# EPICS substitutions: evrMrmApp/Db/evr-pcie-300dc.substitutions
# Record set for a PCIe-EVR-300DC
#
# Macros:
#  EVR = Card name (same as mrmEvrSetupPCI())
#  SYS = System name (ie SR-TM)
#  D = Device name (ie EVR:Diag2)
#  FEVT = Event link frequency (default 124.916 MHz)
#
# Record names have the general forms:
#  $(SYS){$(D)}Signal-SD
#  $(SYS){$(D)-SubDev}Signal-SD

file "evrbase.db"
{
{P="$(SYS){$(D)}", PCNT="$(SYS){$(D)}Cnt:", PLINK="$(SYS){$(D)}Link:", PRATE="$(SYS){$(D)}Rate:", PTIME="$(SYS){$(D)}Time:", OBJ="$(EVR)", OBJBUFRX="$(EVR):BUFRX", EVNT1HZ="\$(EVNT1HZ=125)", FEVT="\$(FEVT=124.916)"}
}

file "databuftx.db"
{pattern
{P, OBJ, PROTO}
{"$(SYS){$(D)}dbus:send:", "$(EVR):BUFTX", 1}
}

file "evrSoftEvt.template"
{
{P="$(SYS){$(D)}", OBJ="$(EVR)"}
}

file "databuftxCtrl.db"
{pattern
{P, OBJ}
{"$(SYS){$(D)}Link:", "$(EVR):BUFTX"}
}

file "mrmevrbufrx.db"
{pattern
{P, OBJ, PROTO}
{"$(SYS){$(D)}dbus:recv:", $(EVR):BUFRX, 0xff00}
}

file mrmSoftSeq.template {
pattern { P, PINITSEQ, PTRIGSRC, EVG, seqNum, NELM }
{ "$(SYS){$(D)-SoftSeq:0}", "$(SYS){$(D)-SoftSeq:0}InitSeq:", "$(SYS){$(D)-SoftSeq:0}TrigSrc:", "$(EVR)", 0, 2047 }
{ "$(SYS){$(D)-SoftSeq:1}", "$(SYS){$(D)-SoftSeq:1}InitSeq:", "$(SYS){$(D)-SoftSeq:1}TrigSrc:", "$(EVR)", 1, 2047 }
{ "$(SYS){$(D)-SoftSeq:2}", "$(SYS){$(D)-SoftSeq:2}InitSeq:", "$(SYS){$(D)-SoftSeq:2}TrigSrc:", "$(EVR)", 2, 2047 }
}

file evrSoftSeq.template {
pattern { P, PTRIGSRC, PEVTCLKFREQ, SYSDEVTCLK, EVG, seqNum, NELM }
{ "$(SYS){$(D)-SoftSeq:0}", "$(SYS){$(D)-SoftSeq:0}TrigSrc:", "$(SYS){$(D)-SoftSeq:0}EvtClkFreq:", "$(SYS){$(D)-EvtClk}", "$(EVR)", 0, 2047 }
{ "$(SYS){$(D)-SoftSeq:1}", "$(SYS){$(D)-SoftSeq:1}TrigSrc:", "$(SYS){$(D)-SoftSeq:1}EvtClkFreq:", "$(SYS){$(D)-EvtClk}", "$(EVR)", 1, 2047 }
{ "$(SYS){$(D)-SoftSeq:2}", "$(SYS){$(D)-SoftSeq:2}TrigSrc:", "$(SYS){$(D)-SoftSeq:2}EvtClkFreq:", "$(SYS){$(D)-EvtClk}", "$(EVR)", 2, 2047 }
}

file "sfp.db"
{
{P="$(SYS){$(D)-SFP}", PPWR="$(SYS){$(D)-SFP}Pwr:", PSPEED="$(SYS){$(D)-SFP}Speed:", PDATE="$(SYS){$(D)-SFP}Date:", OBJ="$(EVR):SFP"}
}

file "mrmevrdc.template"
{
{P="$(SYS){$(D)-DC}", OBJ="$(EVR)"}
}

file "evrmap.db"
{pattern
{NAME, OBJ, func, EVT}
{"$(SYS){$(D)}Evt:Blink0-SP", "$(EVR)", Blink, 15}
{"$(SYS){$(D)}Evt:Blink1-SP", "$(EVR)", Blink, 0}
{"$(SYS){$(D)}Evt:ResetPS-SP","$(EVR)", "Reset PS", 123}
}

file "evrevent.db"
{pattern
{EN, OBJ, CODE, EVNT}
{"$(SYS){$(D)}1hz",  "$(EVR)", 0x7d, 125}
{"$(SYS){$(D)}EvtA", "$(EVR)", 10, 10}
{"$(SYS){$(D)}EvtB", "$(EVR)", 11, 11}
{"$(SYS){$(D)}EvtC", "$(EVR)", 12, 12}
{"$(SYS){$(D)}EvtD", "$(EVR)", 13, 13}
{"$(SYS){$(D)}EvtE", "$(EVR)", 14, 14}
{"$(SYS){$(D)}EvtF", "$(EVR)", 15, 15}
{"$(SYS){$(D)}EvtG", "$(EVR)", 16, 16}
{"$(SYS){$(D)}EvtH", "$(EVR)", 17, 17}
}

file "evrscale.db"
{pattern
{IDX, P, SN, OBJ, MAX}
{0, "$(SYS){$(D)}Link:", "$(SYS){$(D)-PS:$(IDX)}", "$(EVR):PS$(IDX)", "0xffffffff"}
{1, "$(SYS){$(D)}Link:", "$(SYS){$(D)-PS:$(IDX)}", "$(EVR):PS$(IDX)", "0xffffffff"}
{2, "$(SYS){$(D)}Link:", "$(SYS){$(D)-PS:$(IDX)}", "$(EVR):PS$(IDX)", "0xffffffff"}
{3, "$(SYS){$(D)}Link:", "$(SYS){$(D)-PS:$(IDX)}", "$(EVR):PS$(IDX)", "0xffffffff"}
{4, "$(SYS){$(D)}Link:", "$(SYS){$(D)-PS:$(IDX)}", "$(EVR):PS$(IDX)", "0xffffffff"}
{5, "$(SYS){$(D)}Link:", "$(SYS){$(D)-PS:$(IDX)}", "$(EVR):PS$(IDX)", "0xffffffff"}
{6, "$(SYS){$(D)}Link:", "$(SYS){$(D)-PS:$(IDX)}", "$(EVR):PS$(IDX)", "0xffffffff"}
{7, "$(SYS){$(D)}Link:", "$(SYS){$(D)-PS:$(IDX)}", "$(EVR):PS$(IDX)", "0xffffffff"}
}

file "mrmevrout.db"
{pattern
{ON, ONSRC, OBJ, DESC}
{"$(SYS){$(D)-Out:Int}", "$(SYS){$(D)-Out:Int}Src:", "$(EVR):Int", "Internal"}
# default to tri-state for IFB
pattern
{ON, ONSRC, OBJ, DESC, DEFAULT}
{"$(SYS){$(D)-Out:FPUV00}", "$(SYS){$(D)-Out:FPUV00}Src:", "$(EVR):FrontUnivOut0", "UNIV0", 61}
{"$(SYS){$(D)-Out:FPUV01}", "$(SYS){$(D)-Out:FPUV01}Src:", "$(EVR):FrontUnivOut1", "UNIV1", 61}
{"$(SYS){$(D)-Out:FPUV02}", "$(SYS){$(D)-Out:FPUV02}Src:", "$(EVR):FrontUnivOut2", "UNIV2", 61}
{"$(SYS){$(D)-Out:FPUV03}", "$(SYS){$(D)-Out:FPUV03}Src:", "$(EVR):FrontUnivOut3", "UNIV3", 61}
{"$(SYS){$(D)-Out:FPUV04}", "$(SYS){$(D)-Out:FPUV04}Src:", "$(EVR):FrontUnivOut4", "UNIV4", 61}
{"$(SYS){$(D)-Out:FPUV05}", "$(SYS){$(D)-Out:FPUV05}Src:", "$(EVR):FrontUnivOut5", "UNIV5", 61}
{"$(SYS){$(D)-Out:FPUV06}", "$(SYS){$(D)-Out:FPUV06}Src:", "$(EVR):FrontUnivOut6", "UNIV6", 61}
{"$(SYS){$(D)-Out:FPUV07}", "$(SYS){$(D)-Out:FPUV07}Src:", "$(EVR):FrontUnivOut7", "UNIV7", 61}
{"$(SYS){$(D)-Out:FPUV08}", "$(SYS){$(D)-Out:FPUV08}Src:", "$(EVR):FrontUnivOut8", "UNIV8", 61}
{"$(SYS){$(D)-Out:FPUV09}", "$(SYS){$(D)-Out:FPUV09}Src:", "$(EVR):FrontUnivOut9", "UNIV9", 61}
{"$(SYS){$(D)-Out:FPUV10}", "$(SYS){$(D)-Out:FPUV10}Src:", "$(EVR):FrontUnivOut10","UNIV10", 61}
{"$(SYS){$(D)-Out:FPUV11}", "$(SYS){$(D)-Out:FPUV11}Src:", "$(EVR):FrontUnivOut11","UNIV11", 61}
{"$(SYS){$(D)-Out:FPUV12}", "$(SYS){$(D)-Out:FPUV12}Src:", "$(EVR):FrontUnivOut12","UNIV12", 61}
{"$(SYS){$(D)-Out:FPUV13}", "$(SYS){$(D)-Out:FPUV13}Src:", "$(EVR):FrontUnivOut13","UNIV13", 61}
{"$(SYS){$(D)-Out:FPUV14}", "$(SYS){$(D)-Out:FPUV14}Src:", "$(EVR):FrontUnivOut14","UNIV14", 61}
{"$(SYS){$(D)-Out:FPUV15}", "$(SYS){$(D)-Out:FPUV15}Src:", "$(EVR):FrontUnivOut15","UNIV15", 61}
}

file "mrmevroutint.db"
{{
    ON="$(SYS){$(D)-Out:Int}", OBJ="$(EVR)"
}}

# Pulse generators w/o a prescaler set NOPS=1
file "evrpulser.db"
{pattern
{PID, P, PLINK, PN, PNDELAY, PNWIDTH, OBJ, DMAX, WMAX, PMAX, NOPS}
{0, "$(SYS){$(D)}", "$(SYS){$(D)}Link:", "$(SYS){$(D)-DlyGen:$(PID)}", "$(SYS){$(D)-DlyGen:$(PID)}Delay:", "$(SYS){$(D)-DlyGen:$(PID)}Width:", "$(EVR):Pul$(PID)", "0xffffffff", "0xffffffff", "0xffff", 0}
{1, "$(SYS){$(D)}", "$(SYS){$(D)}Link:", "$(SYS){$(D)-DlyGen:$(PID)}", "$(SYS){$(D)-DlyGen:$(PID)}Delay:", "$(SYS){$(D)-DlyGen:$(PID)}Width:", "$(EVR):Pul$(PID)", "0xffffffff", "0xffffffff", "0xffff", 0}
{2, "$(SYS){$(D)}", "$(SYS){$(D)}Link:", "$(SYS){$(D)-DlyGen:$(PID)}", "$(SYS){$(D)-DlyGen:$(PID)}Delay:", "$(SYS){$(D)-DlyGen:$(PID)}Width:", "$(EVR):Pul$(PID)", "0xffffffff", "0xffffffff", "0xffff", 0}
{3, "$(SYS){$(D)}", "$(SYS){$(D)}Link:", "$(SYS){$(D)-DlyGen:$(PID)}", "$(SYS){$(D)-DlyGen:$(PID)}Delay:", "$(SYS){$(D)-DlyGen:$(PID)}Width:", "$(EVR):Pul$(PID)", "0xffffffff", "0xffffffff", "0xffff", 0}
{4, "$(SYS){$(D)}", "$(SYS){$(D)}Link:", "$(SYS){$(D)-DlyGen:$(PID)}", "$(SYS){$(D)-DlyGen:$(PID)}Delay:", "$(SYS){$(D)-DlyGen:$(PID)}Width:", "$(EVR):Pul$(PID)", "0xffffffff", "0xffff", "1", 1}
{5, "$(SYS){$(D)}", "$(SYS){$(D)}Link:", "$(SYS){$(D)-DlyGen:$(PID)}", "$(SYS){$(D)-DlyGen:$(PID)}Delay:", "$(SYS){$(D)-DlyGen:$(PID)}Width:", "$(EVR):Pul$(PID)", "0xffffffff", "0xffff", "1", 1}
{6, "$(SYS){$(D)}", "$(SYS){$(D)}Link:", "$(SYS){$(D)-DlyGen:$(PID)}", "$(SYS){$(D)-DlyGen:$(PID)}Delay:", "$(SYS){$(D)-DlyGen:$(PID)}Width:", "$(EVR):Pul$(PID)", "0xffffffff", "0xffff", "1", 1}
{7, "$(SYS){$(D)}", "$(SYS){$(D)}Link:", "$(SYS){$(D)-DlyGen:$(PID)}", "$(SYS){$(D)-DlyGen:$(PID)}Delay:", "$(SYS){$(D)-DlyGen:$(PID)}Width:", "$(EVR):Pul$(PID)", "0xffffffff", "0xffff", "1", 1}
{8, "$(SYS){$(D)}", "$(SYS){$(D)}Link:", "$(SYS){$(D)-DlyGen:$(PID)}", "$(SYS){$(D)-DlyGen:$(PID)}Delay:", "$(SYS){$(D)-DlyGen:$(PID)}Width:", "$(EVR):Pul$(PID)", "0xffffffff", "0xffff", "1", 1}
{9, "$(SYS){$(D)}", "$(SYS){$(D)}Link:", "$(SYS){$(D)-DlyGen:$(PID)}", "$(SYS){$(D)-DlyGen:$(PID)}Delay:", "$(SYS){$(D)-DlyGen:$(PID)}Width:", "$(EVR):Pul$(PID)", "0xffffffff", "0xffff", "1", 1}
{10,"$(SYS){$(D)}", "$(SYS){$(D)}Link:", "$(SYS){$(D)-DlyGen:$(PID)}", "$(SYS){$(D)-DlyGen:$(PID)}Delay:", "$(SYS){$(D)-DlyGen:$(PID)}Width:", "$(EVR):Pul$(PID)", "0xffffffff", "0xffff", "1", 1}
{11,"$(SYS){$(D)}", "$(SYS){$(D)}Link:", "$(SYS){$(D)-DlyGen:$(PID)}", "$(SYS){$(D)-DlyGen:$(PID)}Delay:", "$(SYS){$(D)-DlyGen:$(PID)}Width:", "$(EVR):Pul$(PID)", "0xffffffff", "0xffff", "1", 1}
{12,"$(SYS){$(D)}", "$(SYS){$(D)}Link:", "$(SYS){$(D)-DlyGen:$(PID)}", "$(SYS){$(D)-DlyGen:$(PID)}Delay:", "$(SYS){$(D)-DlyGen:$(PID)}Width:", "$(EVR):Pul$(PID)", "0xffffffff", "0xffff", "1", 1}
{13,"$(SYS){$(D)}", "$(SYS){$(D)}Link:", "$(SYS){$(D)-DlyGen:$(PID)}", "$(SYS){$(D)-DlyGen:$(PID)}Delay:", "$(SYS){$(D)-DlyGen:$(PID)}Width:", "$(EVR):Pul$(PID)", "0xffffffff", "0xffff", "1", 1}
{14,"$(SYS){$(D)}", "$(SYS){$(D)}Link:", "$(SYS){$(D)-DlyGen:$(PID)}", "$(SYS){$(D)-DlyGen:$(PID)}Delay:", "$(SYS){$(D)-DlyGen:$(PID)}Width:", "$(EVR):Pul$(PID)", "0xffffffff", "0xffff", "1", 1}
{15,"$(SYS){$(D)}", "$(SYS){$(D)}Link:", "$(SYS){$(D)-DlyGen:$(PID)}", "$(SYS){$(D)-DlyGen:$(PID)}Delay:", "$(SYS){$(D)-DlyGen:$(PID)}Width:", "$(EVR):Pul$(PID)", "0xffffffff", "0xffff", "1", 1}
# gate generators
{28,"$(SYS){$(D)}", "$(SYS){$(D)}Link:", "$(SYS){$(D)-DlyGen:$(PID)}", "$(SYS){$(D)-DlyGen:$(PID)}Delay:", "$(SYS){$(D)-DlyGen:$(PID)}Width:", "$(EVR):Pul$(PID)", "0xffffffff", "0xffff", "1", 1}
{29,"$(SYS){$(D)}", "$(SYS){$(D)}Link:", "$(SYS){$(D)-DlyGen:$(PID)}", "$(SYS){$(D)-DlyGen:$(PID)}Delay:", "$(SYS){$(D)-DlyGen:$(PID)}Width:", "$(EVR):Pul$(PID)", "0xffffffff", "0xffff", "1", 1}
{30,"$(SYS){$(D)}", "$(SYS){$(D)}Link:", "$(SYS){$(D)-DlyGen:$(PID)}", "$(SYS){$(D)-DlyGen:$(PID)}Delay:", "$(SYS){$(D)-DlyGen:$(PID)}Width:", "$(EVR):Pul$(PID)", "0xffffffff", "0xffff", "1", 1}
{31,"$(SYS){$(D)}", "$(SYS){$(D)}Link:", "$(SYS){$(D)-DlyGen:$(PID)}", "$(SYS){$(D)-DlyGen:$(PID)}Delay:", "$(SYS){$(D)-DlyGen:$(PID)}Width:", "$(EVR):Pul$(PID)", "0xffffffff", "0xffff", "1", 1}
}

# Default to 3 possible trigger mappings per pulser
file "evrpulsermap.db"
{pattern
{PID, NAME, OBJ, F, EVT}
{0, "$(SYS){$(D)-DlyGen:$(PID)}Evt:Trig0-SP", "$(EVR):Pul$(PID)", Trig, 0}
{0, "$(SYS){$(D)-DlyGen:$(PID)}Evt:Trig1-SP", "$(EVR):Pul$(PID)", Trig, 0}
{0, "$(SYS){$(D)-DlyGen:$(PID)}Evt:Trig2-SP", "$(EVR):Pul$(PID)", Trig, 0}
{1, "$(SYS){$(D)-DlyGen:$(PID)}Evt:Trig0-SP", "$(EVR):Pul$(PID)", Trig, 0}
{1, "$(SYS){$(D)-DlyGen:$(PID)}Evt:Trig1-SP", "$(EVR):Pul$(PID)", Trig, 0}
{1, "$(SYS){$(D)-DlyGen:$(PID)}Evt:Trig2-SP", "$(EVR):Pul$(PID)", Trig, 0}
{2, "$(SYS){$(D)-DlyGen:$(PID)}Evt:Trig0-SP", "$(EVR):Pul$(PID)", Trig, 0}
{2, "$(SYS){$(D)-DlyGen:$(PID)}Evt:Trig1-SP", "$(EVR):Pul$(PID)", Trig, 0}
{2, "$(SYS){$(D)-DlyGen:$(PID)}Evt:Trig2-SP", "$(EVR):Pul$(PID)", Trig, 0}
{3, "$(SYS){$(D)-DlyGen:$(PID)}Evt:Trig0-SP", "$(EVR):Pul$(PID)", Trig, 0}
{3, "$(SYS){$(D)-DlyGen:$(PID)}Evt:Trig1-SP", "$(EVR):Pul$(PID)", Trig, 0}
{3, "$(SYS){$(D)-DlyGen:$(PID)}Evt:Trig2-SP", "$(EVR):Pul$(PID)", Trig, 0}
{4, "$(SYS){$(D)-DlyGen:$(PID)}Evt:Trig0-SP", "$(EVR):Pul$(PID)", Trig, 0}
{4, "$(SYS){$(D)-DlyGen:$(PID)}Evt:Trig1-SP", "$(EVR):Pul$(PID)", Trig, 0}
{4, "$(SYS){$(D)-DlyGen:$(PID)}Evt:Trig2-SP", "$(EVR):Pul$(PID)", Trig, 0}
{5, "$(SYS){$(D)-DlyGen:$(PID)}Evt:Trig0-SP", "$(EVR):Pul$(PID)", Trig, 0}
{5, "$(SYS){$(D)-DlyGen:$(PID)}Evt:Trig1-SP", "$(EVR):Pul$(PID)", Trig, 0}
{5, "$(SYS){$(D)-DlyGen:$(PID)}Evt:Trig2-SP", "$(EVR):Pul$(PID)", Trig, 0}
{6, "$(SYS){$(D)-DlyGen:$(PID)}Evt:Trig0-SP", "$(EVR):Pul$(PID)", Trig, 0}
{6, "$(SYS){$(D)-DlyGen:$(PID)}Evt:Trig1-SP", "$(EVR):Pul$(PID)", Trig, 0}
{6, "$(SYS){$(D)-DlyGen:$(PID)}Evt:Trig2-SP", "$(EVR):Pul$(PID)", Trig, 0}
{7, "$(SYS){$(D)-DlyGen:$(PID)}Evt:Trig0-SP", "$(EVR):Pul$(PID)", Trig, 0}
{7, "$(SYS){$(D)-DlyGen:$(PID)}Evt:Trig1-SP", "$(EVR):Pul$(PID)", Trig, 0}
{7, "$(SYS){$(D)-DlyGen:$(PID)}Evt:Trig2-SP", "$(EVR):Pul$(PID)", Trig, 0}
{8, "$(SYS){$(D)-DlyGen:$(PID)}Evt:Trig0-SP", "$(EVR):Pul$(PID)", Trig, 0}
{8, "$(SYS){$(D)-DlyGen:$(PID)}Evt:Trig1-SP", "$(EVR):Pul$(PID)", Trig, 0}
{8, "$(SYS){$(D)-DlyGen:$(PID)}Evt:Trig2-SP", "$(EVR):Pul$(PID)", Trig, 0}
{9, "$(SYS){$(D)-DlyGen:$(PID)}Evt:Trig0-SP", "$(EVR):Pul$(PID)", Trig, 0}
{9, "$(SYS){$(D)-DlyGen:$(PID)}Evt:Trig1-SP", "$(EVR):Pul$(PID)", Trig, 0}
{9, "$(SYS){$(D)-DlyGen:$(PID)}Evt:Trig2-SP", "$(EVR):Pul$(PID)", Trig, 0}
{10,"$(SYS){$(D)-DlyGen:$(PID)}Evt:Trig0-SP", "$(EVR):Pul$(PID)", Trig, 0}
{10,"$(SYS){$(D)-DlyGen:$(PID)}Evt:Trig1-SP", "$(EVR):Pul$(PID)", Trig, 0}
{10,"$(SYS){$(D)-DlyGen:$(PID)}Evt:Trig2-SP", "$(EVR):Pul$(PID)", Trig, 0}
{11,"$(SYS){$(D)-DlyGen:$(PID)}Evt:Trig0-SP", "$(EVR):Pul$(PID)", Trig, 0}
{11,"$(SYS){$(D)-DlyGen:$(PID)}Evt:Trig1-SP", "$(EVR):Pul$(PID)", Trig, 0}
{11,"$(SYS){$(D)-DlyGen:$(PID)}Evt:Trig2-SP", "$(EVR):Pul$(PID)", Trig, 0}
{12,"$(SYS){$(D)-DlyGen:$(PID)}Evt:Trig0-SP", "$(EVR):Pul$(PID)", Trig, 0}
{12,"$(SYS){$(D)-DlyGen:$(PID)}Evt:Trig1-SP", "$(EVR):Pul$(PID)", Trig, 0}
{12,"$(SYS){$(D)-DlyGen:$(PID)}Evt:Trig2-SP", "$(EVR):Pul$(PID)", Trig, 0}
{13,"$(SYS){$(D)-DlyGen:$(PID)}Evt:Trig0-SP", "$(EVR):Pul$(PID)", Trig, 0}
{13,"$(SYS){$(D)-DlyGen:$(PID)}Evt:Trig1-SP", "$(EVR):Pul$(PID)", Trig, 0}
{13,"$(SYS){$(D)-DlyGen:$(PID)}Evt:Trig2-SP", "$(EVR):Pul$(PID)", Trig, 0}
{14,"$(SYS){$(D)-DlyGen:$(PID)}Evt:Trig0-SP", "$(EVR):Pul$(PID)", Trig, 0}
{14,"$(SYS){$(D)-DlyGen:$(PID)}Evt:Trig1-SP", "$(EVR):Pul$(PID)", Trig, 0}
{14,"$(SYS){$(D)-DlyGen:$(PID)}Evt:Trig2-SP", "$(EVR):Pul$(PID)", Trig, 0}
{15,"$(SYS){$(D)-DlyGen:$(PID)}Evt:Trig0-SP", "$(EVR):Pul$(PID)", Trig, 0}
{15,"$(SYS){$(D)-DlyGen:$(PID)}Evt:Trig1-SP", "$(EVR):Pul$(PID)", Trig, 0}
{15,"$(SYS){$(D)-DlyGen:$(PID)}Evt:Trig2-SP", "$(EVR):Pul$(PID)", Trig, 0}
# gate generators mappings
{28,"$(SYS){$(D)-DlyGen:$(PID)}Evt:Trig0-SP", "$(EVR):Pul$(PID)", Trig, 0}
{28,"$(SYS){$(D)-DlyGen:$(PID)}Evt:Trig1-SP", "$(EVR):Pul$(PID)", Trig, 0}
{28,"$(SYS){$(D)-DlyGen:$(PID)}Evt:Trig2-SP", "$(EVR):Pul$(PID)", Trig, 0}
{29,"$(SYS){$(D)-DlyGen:$(PID)}Evt:Trig0-SP", "$(EVR):Pul$(PID)", Trig, 0}
{29,"$(SYS){$(D)-DlyGen:$(PID)}Evt:Trig1-SP", "$(EVR):Pul$(PID)", Trig, 0}
{29,"$(SYS){$(D)-DlyGen:$(PID)}Evt:Trig2-SP", "$(EVR):Pul$(PID)", Trig, 0}
{30,"$(SYS){$(D)-DlyGen:$(PID)}Evt:Trig0-SP", "$(EVR):Pul$(PID)", Trig, 0}
{30,"$(SYS){$(D)-DlyGen:$(PID)}Evt:Trig1-SP", "$(EVR):Pul$(PID)", Trig, 0}
{30,"$(SYS){$(D)-DlyGen:$(PID)}Evt:Trig2-SP", "$(EVR):Pul$(PID)", Trig, 0}
{31,"$(SYS){$(D)-DlyGen:$(PID)}Evt:Trig0-SP", "$(EVR):Pul$(PID)", Trig, 0}
{31,"$(SYS){$(D)-DlyGen:$(PID)}Evt:Trig1-SP", "$(EVR):Pul$(PID)", Trig, 0}
{31,"$(SYS){$(D)-DlyGen:$(PID)}Evt:Trig2-SP", "$(EVR):Pul$(PID)", Trig, 0}
}

# pulser masking controls
file "evrdcpulser.template"
{pattern
{PID, P, PN, OBJ}
{0, "$(SYS){$(D)}", "$(SYS){$(D)-DlyGen:$(PID)}", "$(EVR):Pul$(PID)"}
{1, "$(SYS){$(D)}", "$(SYS){$(D)-DlyGen:$(PID)}", "$(EVR):Pul$(PID)"}
{2, "$(SYS){$(D)}", "$(SYS){$(D)-DlyGen:$(PID)}", "$(EVR):Pul$(PID)"}
{3, "$(SYS){$(D)}", "$(SYS){$(D)-DlyGen:$(PID)}", "$(EVR):Pul$(PID)"}
{4, "$(SYS){$(D)}", "$(SYS){$(D)-DlyGen:$(PID)}", "$(EVR):Pul$(PID)"}
{5, "$(SYS){$(D)}", "$(SYS){$(D)-DlyGen:$(PID)}", "$(EVR):Pul$(PID)"}
{6, "$(SYS){$(D)}", "$(SYS){$(D)-DlyGen:$(PID)}", "$(EVR):Pul$(PID)"}
{7, "$(SYS){$(D)}", "$(SYS){$(D)-DlyGen:$(PID)}", "$(EVR):Pul$(PID)"}
{8, "$(SYS){$(D)}", "$(SYS){$(D)-DlyGen:$(PID)}", "$(EVR):Pul$(PID)"}
{9, "$(SYS){$(D)}", "$(SYS){$(D)-DlyGen:$(PID)}", "$(EVR):Pul$(PID)"}
{10, "$(SYS){$(D)}", "$(SYS){$(D)-DlyGen:$(PID)}", "$(EVR):Pul$(PID)"}
{11, "$(SYS){$(D)}", "$(SYS){$(D)-DlyGen:$(PID)}", "$(EVR):Pul$(PID)"}
{12, "$(SYS){$(D)}", "$(SYS){$(D)-DlyGen:$(PID)}", "$(EVR):Pul$(PID)"}
{13, "$(SYS){$(D)}", "$(SYS){$(D)-DlyGen:$(PID)}", "$(EVR):Pul$(PID)"}
{14, "$(SYS){$(D)}", "$(SYS){$(D)-DlyGen:$(PID)}", "$(EVR):Pul$(PID)"}
{15, "$(SYS){$(D)}", "$(SYS){$(D)-DlyGen:$(PID)}", "$(EVR):Pul$(PID)"}
}

file "evrin.db"
{pattern
{IN, INTRIG, INCODE, OBJ, DESC}
{"$(SYS){$(D)-In:0}", "$(SYS){$(D)-In:0}Trig:", "$(SYS){$(D)-In:0}Code:", "$(EVR):FPIn0", "IN0 (TTL)"}
{"$(SYS){$(D)-In:1}", "$(SYS){$(D)-In:1}Trig:", "$(SYS){$(D)-In:1}Code:", "$(EVR):FPIn1", "IN1 (TTL)"}
}
